{library PUBLIC}
TYPE DEVICE_TYPE :
(
	TYPE_ERROR:=-1, TYPE_SIMULATED:=0,  TYPE_ABB_1:=1, TYPE_GANTRY_1:=2
);
END_TYPE
//  TYPE_ERROR = '-1'

(* stored: Version 1.1.0.1, ProductVersion 3.1.4024.2
   EnumerationTextList DEVICE_TYPE: Id {9b58185d-b5df-42de-9097-3cac0e44b1e1} *)
